// TIA Portal V20 export
TYPE "typeSequenceControlNode_topTapeAttachment"
// stored: Namespace Unit1.Em3
   STRUCT
      jobs : "LAF_typeJobs";
      sequence : "LAF_typeSequence";
      selectJobStatus { S7_SetPoint := 'True'} : Array[0..10] of "LAF_typeJobStatus";
      "step" : "LER_typeStep";
      jobInterface : "Unit1.Em3.typeSequenceControlNodeJobInterface_topTapeAttachment";
      homeCheck : "Unit1.Em3.typeSequenceControlNodeHomeCheck_topTapeAttachment";
   END_STRUCT;
   // // "step".action1[101] : Step[101] : JOB[1] Condition
   // // "step".action1[110] : Step[110] : Attachment Up
   // // "step".action1[120] : Step[120] : Top Tape X-Axis Remains Attach Pos
   // // "step".action1[130] : Step[130] : Top Tape Attachment Down
   // // "step".action1[140] : Step[140] : Top Tape Attachment Vaccum Off
   // // "step".action1[150] : Step[150] : Top Tape Attachment Up
   // // "step".action1[180] : Step[180] : Top Tape X-Axis Wait Pos
   // // "step".action1[190] : Step[190] : JOB[1] Step End
   // // "step".action1[201] : Step[201] : JOB[2] Condition
   // // "step".action1[210] : Step[210] : Top Tape X-Axis Wait Pos
   // // "step".action1[220] : Step[220] : Top Tape Attachment Down
   // // "step".action1[230] : Step[230] : Top Tape Attachment Vaccum On
   // // "step".action1[240] : Step[240] : Top Tape Cutter Down
   // // "step".action1[241] : Step[241] : Top Tape Cutter Up
   // // "step".action1[242] : Step[242] : Top Tape Clamp Open
   // // "step".action1[250] : Step[250] : Top Tape Attachment Up
   // // "step".action1[290] : Step[290] : JOB[2] Step End
   // // "step".action1[301] : Step[301] : JOB[3] Condition
   // // "step".action1[310] : Step[310] : Top Tape X-Axis Tape-1 Pos
   // // "step".action1[320] : Step[320] : Top Tape Attachment Down
   // // "step".action1[330] : Step[330] : Top Tape Attachment Vaccum Off
   // // "step".action1[370] : Step[370] : Top Tape Attachment Up
   // // "step".action1[380] : Step[380] : Top Tape X-Axis Wait Pos
   // // "step".action1[390] : Step[390] : JOB[3] Step End
   // // "step".action1[401] : Step[401] : JOB[4] Condition
   // // "step".action1[410] : Step[410] : Top Tape X-Axis Tape-2 Pos
   // // "step".action1[420] : Step[420] : Top Tape Attachment Down
   // // "step".action1[430] : Step[430] : Top Tape Attachment Vaccum Off
   // // "step".action1[470] : Step[470] : Top Tape Attachment Up
   // // "step".action1[480] : Step[480] : Top Tape X-Axis Wait Pos
   // // "step".action1[490] : Step[490] : JOB[4] Step End
   // // "step".transition1[101] : Step[101] : JOB[1] Condition
   // // "step".transition1[110] : Step[110] : Attachment Up
   // // "step".transition1[120] : Step[120] : Top Tape X-Axis Remains Attach Pos
   // // "step".transition1[130] : Step[130] : Top Tape Attachment Down
   // // "step".transition1[140] : Step[140] : Top Tape Attachment Vaccum Off
   // // "step".transition1[150] : Step[150] : Top Tape Attachment Up
   // // "step".transition1[180] : Step[180] : Top Tape X-Axis Wait Pos
   // // "step".transition1[190] : Step[190] : JOB[1] Step End
   // // "step".transition1[201] : Step[201] : JOB[2] Condition
   // // "step".transition1[210] : Step[210] : Top Tape X-Axis Wait Pos
   // // "step".transition1[220] : Step[220] : Top Tape Attachment Down
   // // "step".transition1[230] : Step[230] : Top Tape Attachment Vaccum On
   // // "step".transition1[240] : Step[240] : Top Tape Cutter Down
   // // "step".transition1[241] : Step[241] : Top Tape Cutter Up
   // // "step".transition1[242] : Step[242] : Top Tape Clamp Open
   // // "step".transition1[250] : Step[250] : Top Tape Attachment Up
   // // "step".transition1[290] : Step[290] : JOB[2] Step End
   // // "step".transition1[301] : Step[301] : JOB[3] Condition
   // // "step".transition1[310] : Step[310] : Top Tape X-Axis Tape-1 Pos
   // // "step".transition1[320] : Step[320] : Top Tape Attachment Down
   // // "step".transition1[330] : Step[330] : Top Tape Attachment Vaccum Off
   // // "step".transition1[370] : Step[370] : Top Tape Attachment Up
   // // "step".transition1[380] : Step[380] : Top Tape X-Axis Wait Pos
   // // "step".transition1[390] : Step[390] : JOB[3] Step End
   // // "step".transition1[401] : Step[401] : JOB[4] Condition
   // // "step".transition1[410] : Step[410] : Top Tape X-Axis Tape-2 Pos
   // // "step".transition1[420] : Step[420] : Top Tape Attachment Down
   // // "step".transition1[430] : Step[430] : Top Tape Attachment Vaccum Off
   // // "step".transition1[470] : Step[470] : Top Tape Attachment Up
   // // "step".transition1[480] : Step[480] : Top Tape X-Axis Wait Pos
   // // "step".transition1[490] : Step[490] : JOB[4] Step End
END_TYPE
